// TIA Portal V16 export
// export: Created 2021-06-17T11:14:33.8347408Z, ExportSetting WithDefaults, DisplayName Totally Integrated Automation Portal, DisplayVersion V16 Update 4, DisplayName TIA Portal Version Control Interface, DisplayVersion V16 Update 2, DisplayName TIA Portal Openness, DisplayVersion V16 Update 4, DisplayName SINAMICS Startdrive Advanced, DisplayVersion V16 Update 5, DisplayName SINAMICS Startdrive G130, G150, S120, S150, SINAMICS MV, S210, DisplayVersion V16 Update 5, DisplayName SINAMICS Startdrive G110M, G120, G120C, G120D, G120P, G115D, DisplayVersion V16 Update 5, DisplayName STEP 7 Professional, DisplayVersion V16 Update 4, DisplayName SIMATIC Energy Suite, DisplayVersion V16 Update 4, DisplayName STEP 7 Safety, DisplayVersion V16, DisplayName WinCC Advanced / Unified PC, DisplayVersion V16 Update 4, DisplayName SIMATIC Visualization Architect, DisplayVersion V16 Update 1
TYPE "ACB_ETI_HMI"
// stored: IsFailsafeCompliant false
   STRUCT
      QD_ST { ExternalWritable := 'False'} : DWord;   // Status+Mode WORD
      QD_AL { ExternalWritable := 'False'} : DWord;   // Alarm WORD
      QD_EE { ExternalWritable := 'False'} : DWord;   // ExternalError WORD
      QD_IL { ExternalWritable := 'False'} : DWord;   // Interlock WORD
      QI_InterlockedByID { ExternalWritable := 'False'} : Word;   // ID вхідного блокування
      QD_PRM { ExternalWritable := 'False'} : DWord;   // Bit config paremeterts
      QD_ST_SIM { ExternalWritable := 'False'} : DWord;   // Status of Enabled/disabled Simulated parametrs
   END_STRUCT;
END_TYPE
